FUNCTION_BLOCK RunUnitController EXTENDS RunUnitGeneric
VAR_INPUT
END_VAR
VAR_OUTPUT
END_VAR
VAR
	currentMode : eOperationModes := eOperationModes.MANUAL; //default in semi-auto
	
	nCounter : INT;
	bAllInitialized : BOOL := FALSE;
	
	//user control
	requestInitialize : BOOL;
	requestMode : eOperationModes := eOperationModes.SEMI_AUTO;
	//error
	requestErrorClear : eErrorClearWays := eErrorClearWays.NO_ACTION;
	errorDevice : POINTER TO CommonBase := 0; //null reference
	errorType : eCategrories;
	errorIndex : INT;
	errorCode : UDINT;
	errorDelayDetect : TON;
	
	//HMI Control interface
	interfaceControl : InterfaceControlV1;
	interfaceManual : InterfaceManualV1;
	
END_VAR
VAR PERSISTENT
	axisUpperBound : INT;
	cylinderUpperBound : INT;
	signalUpperBound : INT;
	unitUpperBound : INT;
END_VAR

//scan running all devices
FOR nCounter :=1 TO axisUpperBound BY 1 DO
	gvl.axisControls[nCounter]();
	//error detection
	IF errorDevice=0 AND errorDelayDetect.Q AND gvl.axisControls[nCounter].ErrorDetect() <> 0 THEN
		//error scaned
		errorDevice := ADR(gvl.axisControls[nCounter]);
	END_IF
END_FOR
FOR nCounter :=1 TO cylinderUpperBound BY 1 DO
	gvl.cylinderControls[nCounter]();
	//error detection
	IF errorDevice=0 AND errorDelayDetect.Q AND gvl.cylinderControls[nCounter].ErrorDetect() <> 0 THEN
		//error scaned
		errorDevice := ADR(gvl.cylinderControls[nCounter]);
	END_IF
END_FOR
FOR nCounter :=1 TO signalUpperBound BY 1 DO
	gvl.signalControls[nCounter]();
END_FOR
FOR nCounter :=1 TO unitUpperBound BY 1 DO
	//error detection
	IF errorDevice=0 AND errorDelayDetect.Q AND gvl.stations[nCounter] <> 0 AND_THEN gvl.stations[nCounter]^.ErrorDetect() <> 0THEN
		//station
		errorDevice := gvl.stations[nCounter];
	END_IF
END_FOR
//routines
errorDelayDetect(IN:= (errorDevice = 0), PT:= T#100MS, Q=> , ET=> );	//after reset , wait 100ms to detect
IF errorDevice <>0 THEN
	errorIndex := nCounter-1;
	errorType := errorDevice^.TypeCode();
	errorCode := errorDevice^.ErrorDetect();
		
	THIS^.ErrorHandler();// handling user-input reset/ignore
END_IF
//reflect to interface
//
interfaceManual(
	currentMode:= THIS^.currentMode); //scan-in,scan-out,manual...
//handling input request
interfaceControl(
	currentMode:= THIS^.currentMode, 
	requestMode=> THIS^.requestMode, 
	errorClear=> THIS^.requestErrorClear, 
	mMonitorDatas=> );
IF interfaceControl.requestInit THEN
	requestInitialize := TRUE; // memorize
END_IF	
//mode switcher pre-check
bPause := NOT (currentMode = eOperationModes.AUTO);
IF requestMode<>currentMode THEN
	CASE requestMode OF 
		eOperationModes.MANUAL,eOperationModes.SEMI_AUTO:
			//direct changes
			currentMode := requestMode;
		eOperationModes.AUTO:
			//check : no error , manual channel work done
			IF errorDevice=0 THEN
				currentMode := eOperationModes.AUTO;
			ELSE
				//refuce to change , maintain
				requestMode := currentMode;
			END_IF 
	END_CASE
END_IF
//
CASE currentMode OF	
		eOperationModes.AUTO,eOperationModes.SEMI_AUTO:
		//running sequences
		FOR nCounter :=1 TO unitUpperBound BY 1 DO
			IF gvl.stations[nCounter] <> 0 THEN
				gvl.stations[nCounter]^();
			END_IF
		END_FOR
		
		IF  requestInitialize THEN
			//initialize all stations
			bAllInitialized := TRUE;
			FOR nCounter:=1 TO unitUpperBound BY 1 DO
				IF gvl.stations[nCounter] <> 0 THEN
					// if every station comes initialized
					bAllInitialized := bAllInitialized AND gvl.stations[nCounter]^.Initialize();
				END_IF
			END_FOR
			IF bAllInitialized THEN
				FOR nCounter:=1 TO unitUpperBound BY 1 DO
					IF gvl.stations[nCounter] <> 0 THEN
						gvl.stations[nCounter]^.NextState := 0; //start working
					END_IF
				END_FOR	
				requestInitialize := FALSE; //clear after done
			END_IF
		END_IF		
END_CASE

METHOD ErrorHandler : BOOL
VAR_INPUT
END_VAR
VAR
END_VAR
//once error scanned
IF requestMode = eOperationModes.AUTO THEN
	//once error deteted and in AUTO mode , forcely switch to SEMI_AUTO
	requestMode := eOperationModes.SEMI_AUTO;
END_IF
//reset error handling
IF requestErrorClear <> eErrorClearWays.NO_ACTION THEN
	errorDevice^.ErrorClear(requestErrorClear);
	requestErrorClear := eErrorClearWays.NO_ACTION;
	errorDevice := 0 ;// cut link
END_IF
END_METHOD

METHOD Initialize : BOOL
VAR_INPUT
END_VAR
END_METHOD

END_FUNCTION_BLOCK

(* stored: Version 1.1.0.1, ProductVersion 3.1.4022.10
   POU RunUnitController: Id {dbefb355-befd-4ccc-b7d8-49a15cbd5d5f}, SpecialFunc None
   Method ErrorHandler: Id {a0eb5aec-6465-4175-9953-8d5b0f3a2dc2}
   Method Initialize: Id {cb68dc91-f1ca-48a3-a360-7027131d9307} *)
